GLOBALCONSTANTS IG1_NAME_Functions (* Industry Group 1 specific function defines *)
  (* Standard: 61499-1 *)
  (* Version 1.0, 2026-06-29, Franz Höpfinger, Demmler Andreas Fahrzeugbau *)
  PACKAGE isobus::pgn::const;
  VAR_GLOBAL CONSTANT
    F_TACHOGRAPH : BYTE := 128; (* Sys: Non-specific System, Func: Tachograph *)
    F_DOOR_CONTROLLER : BYTE := 129; (* Sys: Non-specific System, Func: Door Controller *)
    F_ARTICULATION_TURNTABLE_CONTROL : BYTE := 130; (* Sys: Non-specific System, Func: Articulation Turntable Control - Control of the articulation *)
    F_BODY_TO_VEHICLE_INTERFACE_CONTROL : BYTE := 131; (* Sys: Non-specific System, Func: Body-to-Vehicle Interface Control - Interface controller managing *)
    F_SLOPE_SENSOR : BYTE := 132; (* Sys: Non-specific System, Func: Slope Sensor - Sensor for measuring a slope along an axis. *)
    F_RETARDER_DISPLAY : BYTE := 134; (* Sys: Non-specific System, Func: Retarder Display - Display module that shows information *)
    F_DIFFERENTIAL_LOCK_CONTROLLER : BYTE := 135; (* Sys: Non-specific System, Func: Differential Lock Controller *)
    F_LOW_VOLTAGE_DISCONNECT : BYTE := 136; (* Sys: Non-specific System, Func: Low-Voltage Disconnect - The device that monitors the voltage of *)
    F_ROADWAY_INFORMATION : BYTE := 137; (* Sys: Non-specific System, Func: Roadway Information - Devices that use this function will provide *)
    F_AUTOMATED_DRIVING : BYTE := 138; (* Sys: Non-specific System, Func: Automated Driving - Automated Driving System. Note: The hardware *)
    F_NOT_AVAILABLE : BYTE := 255; (* Sys: Non-specific System, Func: Not Available - This assignment can be used until an explicit *)
    F_TRACTOR_FORWARD_ROAD_IMAGE_PROCESSING : BYTE := 128; (* Sys: Tractor, Func: Forward Road Image Processing - Determine vehicle position from lane *)
    F_TRACTOR_FIFTH_WHEEL_SMART_SYSTEM : BYTE := 129; (* Sys: Tractor, Func: Fifth Wheel Smart System - Any systems relative to the operation & *)
    F_TRACTOR_CATALYST_FLUID_SENSOR : BYTE := 130; (* Sys: Tractor, Func: Catalyst Fluid Sensor - The Catalyst Fluid Sensor can measure the catalyst *)
    F_TRACTOR_ADAPTIVE_FRONT_LIGHTING_SYSTEM : BYTE := 131; (* Sys: Tractor, Func: Adaptive Front Lighting System - System used to adjust the vehicle front *)
    F_TRACTOR_IDLE_CONTROL_SYSTEM : BYTE := 132; (* Sys: Tractor, Func: Idle Control System - The device automatically starts and stops the engine *)
    F_TRACTOR_USER_INTERFACE_SYSTEM : BYTE := 133; (* Sys: Tractor, Func: User Interface System - The User Interface System is a two way interface *)
    F_TRACTOR_NOT_AVAILABLE : BYTE := 255; (* Sys: Tractor, Func: Not Available - This assignment can be used until an explicit function has *)
    F_TRAILER_NOT_AVAILABLE : BYTE := 255; (* Sys: Trailer, Func: Not Available - This assignment can be used until an explicit function has *)
  END_VAR
END_GLOBALCONSTANTS
